PROGRAM MAIN
VAR

END_VAR

CallStandardModule();
CallStandard();

END_PROGRAM

(* stored: Version 1.1.0.1, ProductVersion 3.1.4024.12
   POU MAIN: Id {bcf86dc7-f00c-42de-a2d5-2496793eff91}, SpecialFunc None *)
